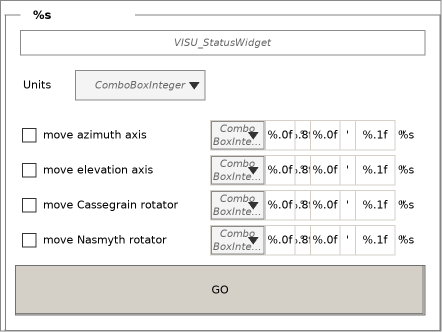
VISUALIZATION VISU_AxesMultiMoveProcess  // 442x332
VAR_IN_OUT
	ref : AxesMultiMoveProcess;
    widget : AxesMultiMoveProcessWidget;
END_VAR
    Polyline (20,15) (5,15) (5,330) (440,330) (440,15) (135,15)
    Label (20,70 80x30), "Units"
    ComboBoxInteger (75,70 130x30), variable: widget.units, text list: 'AxesMoveProcessUnitsTextList'
    Rectangle (395,120 35x30), "%s", text variable: widget.unitsText, invisible if: widget.units = AxesMoveProcessWidgetUnits.DEGMINSEC
    Checkbox (20,120 180x30), "move azimuth axis", variable: widget.selected_azi
    Textfield (210,120 180x30), "%.8f", text variable: widget.field_azi_decimal, invisible if: widget.units = AxesMoveProcessWidgetUnits.DEGMINSEC
        OnMouseClick: write the text variable via VisuDialogs.Numpad
    Textfield (265,120 30x30), "%.0f", text variable: widget.field_azi_d, invisible if: widget.units <> AxesMoveProcessWidgetUnits.DEGMINSEC
        OnMouseClick: write the text variable via VisuDialogs.Numpad
    ComboBoxInteger (211,121 53x28), variable: widget.field_azi_sign, invisible if: widget.units <> AxesMoveProcessWidgetUnits.DEGMINSEC, text list: 'AxesDialogSignTextList'
    Textfield (310,120 30x30), "%.0f", text variable: widget.field_azi_m, invisible if: widget.units <> AxesMoveProcessWidgetUnits.DEGMINSEC
        OnMouseClick: write the text variable via VisuDialogs.Numpad
    Textfield (355,120 40x30), "%.1f", text variable: widget.field_azi_s, invisible if: widget.units <> AxesMoveProcessWidgetUnits.DEGMINSEC
        OnMouseClick: write the text variable via VisuDialogs.Numpad
    Label (295,120 15x30), "°", invisible if: widget.units <> AxesMoveProcessWidgetUnits.DEGMINSEC
    Label (340,120 15x30), "'", invisible if: widget.units <> AxesMoveProcessWidgetUnits.DEGMINSEC
    Label (395,120 15x30), """, invisible if: widget.units <> AxesMoveProcessWidgetUnits.DEGMINSEC
    Button (15,265 410x50), "GO", input disabled if: ref.statuses.enabledStatus.disabled
        OnMouseClick: execute {
            ref.request(
                units := AxesMoveUnits.DEGREES,
                azi := widget.aziDeg,
                ele := widget.eleDeg,
                rot := 0.0,
                roc := widget.rocDeg,
                ron := widget.ronDeg,
                doAzi := widget.selected_azi,
                doEle := widget.selected_ele,
                doRot := FALSE,
                doRoc := widget.selected_roc,
                doRon := widget.selected_ron,
                preferMostTravel := FALSE);
        }
    Checkbox (20,190 185x30), "move Cassegrain rotator", variable: widget.selected_roc
    Checkbox (20,225 175x30), "move Nasmyth rotator", variable: widget.selected_ron
    Checkbox (20,155 180x30), "move elevation axis", variable: widget.selected_ele
    Rectangle (395,155 35x30), "%s", text variable: widget.unitsText, invisible if: widget.units = AxesMoveProcessWidgetUnits.DEGMINSEC
    Textfield (210,155 180x30), "%.8f", text variable: widget.field_ele_decimal, invisible if: widget.units = AxesMoveProcessWidgetUnits.DEGMINSEC
        OnMouseClick: write the text variable via VisuDialogs.Numpad
    Textfield (265,155 30x30), "%.0f", text variable: widget.field_ele_d, invisible if: widget.units <> AxesMoveProcessWidgetUnits.DEGMINSEC
        OnMouseClick: write the text variable via VisuDialogs.Numpad
    ComboBoxInteger (211,156 53x28), variable: widget.field_ele_sign, invisible if: widget.units <> AxesMoveProcessWidgetUnits.DEGMINSEC, text list: 'AxesDialogSignTextList'
    Textfield (310,155 30x30), "%.0f", text variable: widget.field_ele_m, invisible if: widget.units <> AxesMoveProcessWidgetUnits.DEGMINSEC
        OnMouseClick: write the text variable via VisuDialogs.Numpad
    Textfield (355,155 40x30), "%.1f", text variable: widget.field_ele_s, invisible if: widget.units <> AxesMoveProcessWidgetUnits.DEGMINSEC
        OnMouseClick: write the text variable via VisuDialogs.Numpad
    Label (295,155 15x30), "°", invisible if: widget.units <> AxesMoveProcessWidgetUnits.DEGMINSEC
    Label (340,155 15x30), "'", invisible if: widget.units <> AxesMoveProcessWidgetUnits.DEGMINSEC
    Label (395,155 15x30), """, invisible if: widget.units <> AxesMoveProcessWidgetUnits.DEGMINSEC
    Rectangle (395,190 35x30), "%s", text variable: widget.unitsText, invisible if: widget.units = AxesMoveProcessWidgetUnits.DEGMINSEC
    Textfield (210,190 180x30), "%.8f", text variable: widget.field_roc_decimal, invisible if: widget.units = AxesMoveProcessWidgetUnits.DEGMINSEC
        OnMouseClick: write the text variable via VisuDialogs.Numpad
    Textfield (265,190 30x30), "%.0f", text variable: widget.field_roc_d, invisible if: widget.units <> AxesMoveProcessWidgetUnits.DEGMINSEC
        OnMouseClick: write the text variable via VisuDialogs.Numpad
    ComboBoxInteger (211,191 53x28), variable: widget.field_roc_sign, invisible if: widget.units <> AxesMoveProcessWidgetUnits.DEGMINSEC, text list: 'AxesDialogSignTextList'
    Textfield (310,190 30x30), "%.0f", text variable: widget.field_roc_m, invisible if: widget.units <> AxesMoveProcessWidgetUnits.DEGMINSEC
        OnMouseClick: write the text variable via VisuDialogs.Numpad
    Textfield (355,190 40x30), "%.1f", text variable: widget.field_roc_s, invisible if: widget.units <> AxesMoveProcessWidgetUnits.DEGMINSEC
        OnMouseClick: write the text variable via VisuDialogs.Numpad
    Label (295,190 15x30), "°", invisible if: widget.units <> AxesMoveProcessWidgetUnits.DEGMINSEC
    Label (340,190 15x30), "'", invisible if: widget.units <> AxesMoveProcessWidgetUnits.DEGMINSEC
    Label (395,190 15x30), """, invisible if: widget.units <> AxesMoveProcessWidgetUnits.DEGMINSEC
    Rectangle (395,225 35x30), "%s", text variable: widget.unitsText, invisible if: widget.units = AxesMoveProcessWidgetUnits.DEGMINSEC
    Textfield (210,225 180x30), "%.8f", text variable: widget.field_ron_decimal, invisible if: widget.units = AxesMoveProcessWidgetUnits.DEGMINSEC
        OnMouseClick: write the text variable via VisuDialogs.Numpad
    Textfield (265,225 30x30), "%.0f", text variable: widget.field_ron_d, invisible if: widget.units <> AxesMoveProcessWidgetUnits.DEGMINSEC
        OnMouseClick: write the text variable via VisuDialogs.Numpad
    ComboBoxInteger (211,226 53x28), variable: widget.field_ron_sign, invisible if: widget.units <> AxesMoveProcessWidgetUnits.DEGMINSEC, text list: 'AxesDialogSignTextList'
    Textfield (310,225 30x30), "%.0f", text variable: widget.field_ron_m, invisible if: widget.units <> AxesMoveProcessWidgetUnits.DEGMINSEC
        OnMouseClick: write the text variable via VisuDialogs.Numpad
    Textfield (355,225 40x30), "%.1f", text variable: widget.field_ron_s, invisible if: widget.units <> AxesMoveProcessWidgetUnits.DEGMINSEC
        OnMouseClick: write the text variable via VisuDialogs.Numpad
    Label (295,225 15x30), "°", invisible if: widget.units <> AxesMoveProcessWidgetUnits.DEGMINSEC
    Label (340,225 15x30), "'", invisible if: widget.units <> AxesMoveProcessWidgetUnits.DEGMINSEC
    Label (395,225 15x30), """, invisible if: widget.units <> AxesMoveProcessWidgetUnits.DEGMINSEC
    Frame (20,30 405x25)
        shows VISU_StatusWidget(widget := widget.actualStatus)
    Rectangle (30,0 115x30), "%s", text variable: widget.title
END_VISUALIZATION

(* stored: Version 1.1.0.1, ProductVersion 3.1.4019.2
   Visu VISU_AxesMultiMoveProcess: Id {ddfd81e8-b381-4928-9ef1-9c8721259a1c} *)
